TYPE printLogModule_EX_DataST :
STRUCT
	sTime			:WSTRING(255);
	msg				:WSTRING(255);//T_MaxString
END_STRUCT
END_TYPE

(* stored: Version 1.1.0.1, ProductVersion 3.1.4024.4
   DUT printLogModule_EX_DataST: Id {a2c1c46a-908d-4d1a-a0b2-a40896cceef0} *)
